// Mitsubishi GX Works2 project: Lab_2_insys_gxkode   PLC: FX1N/FX1NC

// global labels: Global1
VAR_GLOBAL
  Stopp AT X002 : BOOL;  (* holdekontakt, så lav betyr at den skal stoppes *)
  start_medurs AT X001 : BOOL;
  start_moturs AT X000 : BOOL;
  motorvern AT X003 : BOOL;
  På_lampe AT Y000 : BOOL;
  medurs_lampe AT Y001 : BOOL;
  moturs_lampe AT Y002 : BOOL;
  medurs AT Y003 : BOOL;
  moturs AT Y004 : BOOL;
  hold_kontakt_timer_1 : BOOL;
  hold_kontakt_timer_2 : BOOL;
  prev_dir : BOOL;
  retningsbytte : BOOL;
END_VAR

// task Task_01 (event TRUE, interval 0, priority 31): Lab_2_dreieretning

PROGRAM Lab_2_dreieretning
(* structured ladder/FBD written out as ST: instructions are called as NAME(EN, inputs, outputs); _pN, _eN, _tN stand for wires *)
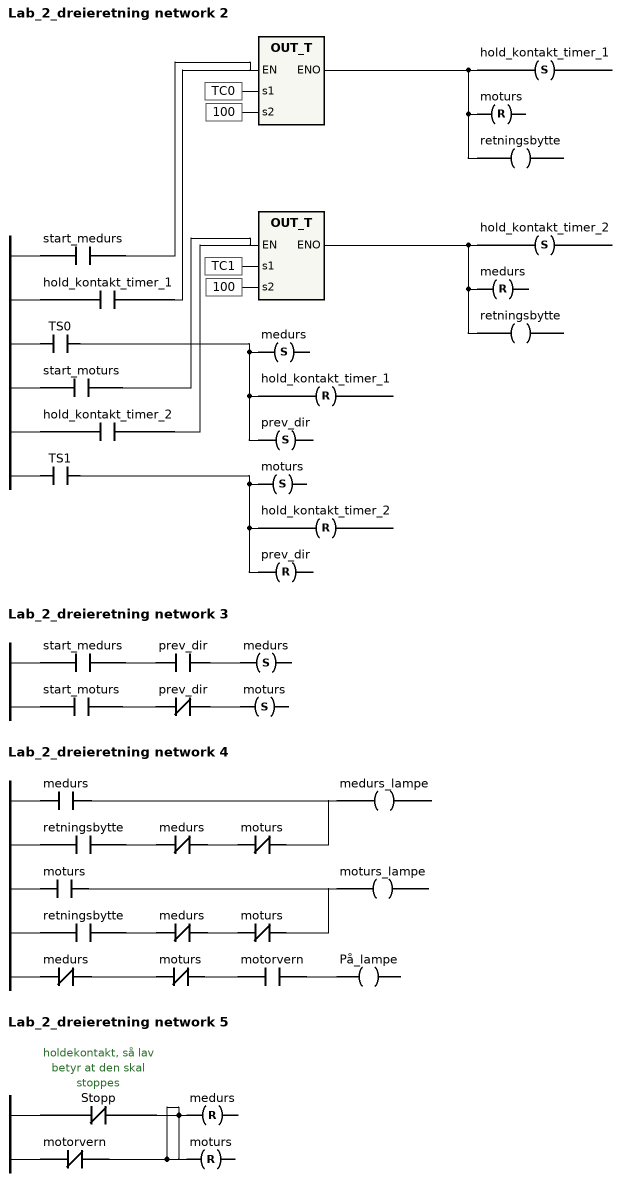
(* network 2 *)
_e1 := OUT_T(start_medurs OR hold_kontakt_timer_1, TC0, 100);
SET(_e1, hold_kontakt_timer_1);
RST(_e1, moturs);
retningsbytte := _e1;
SET(TS0, medurs);
RST(TS0, hold_kontakt_timer_1);
SET(TS0, prev_dir);
_e2 := OUT_T(start_moturs OR hold_kontakt_timer_2, TC1, 100);
SET(_e2, hold_kontakt_timer_2);
RST(_e2, medurs);
SET(TS1, moturs);
retningsbytte := _e2;
RST(TS1, hold_kontakt_timer_2);
RST(TS1, prev_dir);
(* network 3 *)
SET(start_medurs AND prev_dir, medurs);
SET(start_moturs AND NOT prev_dir, moturs);
(* network 4 *)
medurs_lampe := medurs OR (retningsbytte AND NOT medurs AND NOT moturs);
moturs_lampe := moturs OR (retningsbytte AND NOT medurs AND NOT moturs);
På_lampe := NOT medurs AND NOT moturs AND motorvern;
(* network 5 *)
_p1 := (NOT Stopp) OR (NOT motorvern);
RST(_p1, medurs);
RST(_p1, moturs);
END_PROGRAM
